{attribute 'qualified_only'}
VAR_GLOBAL
	MotorActive AT %Q* : BOOL;
	StartMotor AT %I* : BOOL;
	StopMotor AT %I* : BOOL;
END_VAR

(* stored: Version 1.1.0.1, ProductVersion 3.1.4024.12
   GVL GVL: Id {b5db8d1c-63aa-412a-b4aa-18b564493082} *)
